(* CoDeSys 2.3 export: PLC_PRG.EXP *)

(* POU PLC_PRG, ST *)
PROGRAM PLC_PRG
VAR
END_VAR
Read_Inputs;

Write_Outputs;
END_PROGRAM
